TYPE BitStruct : STRUCT
    bBit0 : BIT;
    bBit1 : BIT;
    bBit2 : BIT;
    bBit3 : BIT;
    bBit4 : BIT;
    bBit5 : BIT;
    bBit6 : BIT;
    bBit7 : BIT;
END_STRUCT
END_TYPE

(* stored: Version 1.1.0.1, ProductVersion 3.1.4024.12
   DUT BitStruct: Id {87e02438-32aa-0583-2163-80d88d401a23} *)
